# EPICS autosave request: ipApp/Db/PTC10_rtd_chan_settings.req
$(P)$(T):$(C):temperature.SCAN
#$(P)$(T):$(C):sensor
$(P)$(T):$(C):range
$(P)$(T):$(C):current
$(P)$(T):$(C):power
